(* IEC 61131-3 sources: automatisme-pour-robotique/02_TP/TP_02, 5 files *)

(* ---- HMI_types_FB.st ---- *)
TYPE THmi
    STRUCT
        m_Inputs : THmiInputs ;
        m_Outputs : THmiOutputs ;
    END_STRUCT
END_TYPE

(* ---- TCtrlStatusGroup.st ---- *)
TYPE TCtrlStatusGroup
    STRUCT
        m_xEnable : BOOL ;
        m_xBusy : BOOL ;
        m_xDone : BOOL ;
        m_xError : BOOL ;
        m_udiErrorID : UDINT ;
        m_xTimeOut : BOOL ;
    END_STRUCT
END_TYPE

(* ---- types_staubli.st ---- *)
TYPE T_StaeubliRobot :
    STRUCT
        Status : T_Status ;
        Command : T_Command ;
        CommandInterface : T_CommandInterface ;
    END_STRUCT
END_TYPE

TYPE T_Status:
    STRUCT
        Initialized: BOOL ; (* True = The library is initialized *)
        Online: BOOL ; (* True = robot can receive commands *)
        ErrorPending: BOOL ; (* True = an error is pending *)
        IsMoving: BOOL ; (* True = robot is moving *)
        EStopActive: BOOL ; (* True = E-stop is pending *)
        DummyPlug: BOOL ; (* True = staubli teach pendant replaced by dummy
        plug *)
        ExternalMcp_Wms: BOOL ; (* True = Robot is properly configured to use both
        user- supplied WMS and Teach Pendant. *)
        ActualSpeed: REAL ; (* Cartesian speed of the current TCP *)
        ActualOverride: REAL ; (* Current override value [0.01 .. 100] *)
        ActualErrorNumber: UINT ; (* Total number of pending errors in robot *)
        ActualOperationMode: UINT ; (* Actual working mode 0= invalid , 1=manu,
        3=Auto, 4=remote(extaut) *)
        ActualErrorID: T_PendingErrors ; (* List of pending error on server side *)
        CartesianPos: T_CartesianPos ; (* Current cartesian position *)
        JointPos: T_JointPos ; (* Current joint position *)
        ActualCoordSystem: UINT ; (* Number of the user frame in which the position of
        the Tool Center Point is reported *)
        ActualTool: UINT ; (* Number of the Tool Center Point for which the
        position is reported *)
        RobotStateMachine: UINT ; (* State Machine of the robot *)
        MovementID: INT ; (* Identifier of motion currently executed *)
        MovementProgress: INT ; (* Percentage of actual movement that has been
        completed *)
        RobotModel: INT (* Robot model connected to controller *)
        ControllerModel: UINT ; (* Staubli controller 8=CS8C / 9=CS9 *)
        CS9Safety: T_CS9SftyFbk ; (* CS9 Only - Safety features *)
        Heartbeat: UINT ;
        ServerMajorVersion: UINT ; (* Major version of unival PLC server *)
        ServerMinorVersion: UINT ; (* Minor version of unival PLC server *)
        ServerEdit: UINT ; (* Edit of the uniVAL plc server *)
        ClientMajorVersion: UINT ; (* Major version of unival PLC client library *)
        ClientMinorVersion: UINT ; (* Minor version of unival PLC client library *)
        ClientEdit: UINT ; (* Edit of the unival PLC client library *)
    END_STRUCT
END_TYPE

TYPE T_Command :
    STRUCT
        EnableVerbose : BOOL ; (* TRUE=Enable tracing activity of the server. It is
        strongly recommended to enable trace for debugging
        purpose only. Starting with FALSE *)
        OverrideCmd : UINT ; (* Commanded Override [1..100] (monitor speed) Starting
        with 0 *)
        OperationModeCmd : UINT ; (* Commanded operation mode 0= invalid , 1= Manu,
        3=Auto, 4 remote(extAut) *)
        ToolCmd : UINT ; (* Select the Tool used for movement. Starting with 0*)
        CoordSystemCmd : UINT ; (* Select the coordinate system used for movement.
        Starting with 0 *)
        CS9Safety : T_CS9SftyCmd ; (* CS9 Only - Safety features *)
        LifebitPeriod : TIME ; (* Select the period of the internal lifebit
        (100ms<Period<1000ms) . starting with t#200ms *)
    END_STRUCT
END_TYPE

(* ---- FB_Staubli.st ---- *)
FUNCTION_BLOCK VAL_ReadAxesGroup
    VAR_INPUT
        Enable : BOOL ; (* TRUE : contents of the FB is executed *)
    END_VAR
    VAR_IN_OUT
        AxesGroup : T_StaeubliRobot ; (* Data block for a robot *)
        IN : T_FromRobot ;
    END_VAR
    VAR_OUTPUT
        Error : BOOL ; (* set when function block has terminated with error *)
        ErrorID : UDINT ; (* error code *)
        Timeout : BOOL ; (* set when a timeout is detected *)
    END_VAR

FUNCTION_BLOCK VAL_WriteAxesGroup
    VAR_INPUT
        Enable : BOOL ; (TRUE : contents of the FB is executed *)
    END_VAR
    VAR_IN_OUT
        AxesGroup : T_StaeubliRobot ; (* Data block for a robot *)
    END_VAR
    VAR_OUTPUT
        Error : BOOL ; (* set when function block has terminated with error *)
        ErrorID : UDINT ; (* error code *)
        OUT : T_ToRobot ;
        Timeout : BOOL ; (* set when a timeout is detected *)
    END_VAR

(* ---- FB_VAL_ReadWriteIO.st ---- *)
FUNCTION_BLOCK VAL_ReadWriteIO
    (* Update the digital outputs of the controller with values passed as parameter.
    Return the state of the digital inputs available on the controller *)
    VAR_INPUT
        Enable : BOOL ; (*function block content is executed as long as this input is TRUE *)
        Valve1 : BOOL ; (* 6 axis robot only : the internal valve *)
        Valve2 : BOOL ; (* 6 axis robot only : the internal valve *)
        Fout0 : BOOL ; (* Command Fast output (J212-4 / J212-9) CS9 controller *)
        Fout1 : BOOL ; (* Command Fast output (J212-1 / J212-5) CS9 controller *)
        EnableValve1 : BOOL ; (* 6 axis robot only : the internal valve 5-3 closed middle *)
        EnableValve2 : BOOL ; (* 6 axis robot only : the internal valve 5-3 closed middle *)
    END_VAR
    VAR_IN_OUT
        AxesGroup : T_StaeubliRobot; (* Data block for a robot *)
    END_VAR
    VAR_OUTPUT
        Valid : BOOL ; (*Set when function block is executing. Reset when Done or Error*)
        UsrInput0 : BOOL ; (* Digital input (J109-11 / J109-30) CS8 controller *)
        UsrInput1 : BOOL ; (* Digital input (J109-16 / J109-35) CS8 controller *)
        Fin0 : BOOL ; (* Fast input (J111-2/7) CS8 controller, J212-2/7 CS9 controller *)
        Fin1 : BOOL ; (* Fast input (J111-3/8) CS8 controller, J212-3/8 CS9 controller *)
        ValvesSafeState : BOOL ; (* CS9 controlling 5-3 ways valves ONLY *)
    END_VAR
